TYPE IO :
STRUCT
MesEventCode : ARRAY[1..7] OF WORD ; (*Akuo AlarmCode*)

END_STRUCT
END_TYPE

(* stored: Version 1.1.0.1, ProductVersion 3.1.4024.6
   DUT IO: Id {75a990db-ddee-4d68-8294-db7de02acc22} *)
